ABB RobotStudio station: Robot Manipulatin Assignment 2 task 2.rspag

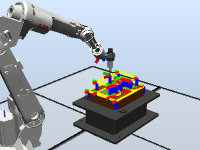
--- station ---
Station try1 (saved by RobotStudio 6.8.8148.134)
Controller IRB_1520ID_4kg_1.50m
  mechanical unit ROB_1: IRB1520ID_4_150__02, 6 joints, base frame (0, 0, 0) mm
Layout (positions relative to the parent item):
  - IRB1520ID_4_150__02 [mechanism, from Robots\IRB1520ID_4_150_G_02.rslib] at (0, 0, 0) mm; joint values [-0.2556, -0.3637, 0.7959, 0.3224, 0.5136, -0.4862] (rad or m)
  - MyTool [mechanism, from Training Objects\myTool.rslib] at (791.12, -174.55, 725.53) mm, rotated rx 180 ry 38 rz 180 deg
  - Robotpedestal1400_H240 [part, from Equipment\Robot Pedestal 1400 H240.rslib] at (1106.08, -98.58, 0) mm
  - Curve_thing [part, from Training Objects\Curve_Thing.rslib] at (902, -245, 225) mm
  - Frame_1 [frame] at (902, -245, 225) mm
Attachment: MyTool is attached to IRB1520ID_4_150__02 / Link6

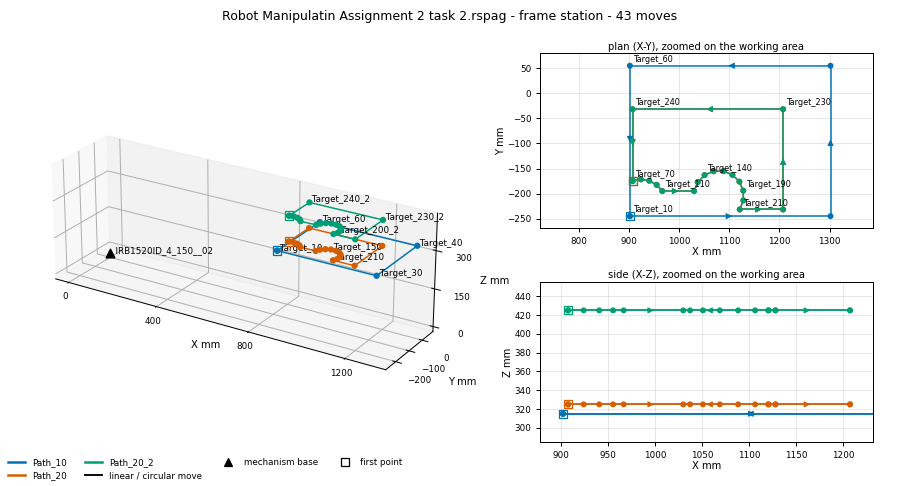
[picture p0: tool path of Robot Manipulatin Assignment 2 task 2.rspag in frame station, 43 of 49 moves have a stored position in this frame; points joined in program order, loops and branches not executed]
--- Backups/IRB_1520ID_4kg_1.50m/RAPID/TASK1/PROGMOD/CalibData.mod ---
MODULE CalibData
	PERS tooldata MyTool:=[TRUE,[[31.792631019,0,229.638935148],[0.945518576,0,0.325568154,0]],[1,[0,0,1],[1,0,0,0],0,0,0]];
ENDMODULE

--- Backups/IRB_1520ID_4kg_1.50m/RAPID/TASK1/PROGMOD/Module1.mod ---
MODULE Module1
    CONST robtarget Target_10:=[[901.999,-245.004,315],[0,0,1,0],[0,0,0,0],[9E+09,9E+09,9E+09,9E+09,9E+09,9E+09]];
    CONST robtarget Target_30:=[[1301.999,-245.004,315],[0,0,1,0],[0,0,0,0],[9E+09,9E+09,9E+09,9E+09,9E+09,9E+09]];
    CONST robtarget Target_40:=[[1301.999,54.996,315],[0,0,1,0],[0,0,0,0],[9E+09,9E+09,9E+09,9E+09,9E+09,9E+09]];
    CONST robtarget Target_60:=[[901.999,54.996,315],[0,0,1,0],[0,0,0,0],[9E+09,9E+09,9E+09,9E+09,9E+09,9E+09]];
    CONST robtarget Target_70:=[[907.446746826,-174.551583792,325],[0,0,1,0],[0,0,0,0],[9E+09,9E+09,9E+09,9E+09,9E+09,9E+09]];
    CONST robtarget Target_80:=[[924.004893302,-171.650689779,325],[0,0,1,0],[0,0,0,0],[9E+09,9E+09,9E+09,9E+09,9E+09,9E+09]];
    CONST robtarget Target_90:=[[940.588636002,-174.40148582,325],[0,0,1,0],[0,0,0,0],[9E+09,9E+09,9E+09,9E+09,9E+09,9E+09]];
    CONST robtarget Target_100:=[[955.323432229,-182.493035793,325],[0,0,1,0],[0,0,0,0],[9E+09,9E+09,9E+09,9E+09,9E+09,9E+09]];
    CONST robtarget Target_110:=[[966.543734874,-195.01071167,325],[0,0,1,0],[0,0,0,0],[9E+09,9E+09,9E+09,9E+09,9E+09,9E+09]];
    CONST robtarget Target_120:=[[1029.963932921,-195.01071167,325],[0,0,1,0],[0,0,0,0],[9E+09,9E+09,9E+09,9E+09,9E+09,9E+09]];
    CONST robtarget Target_130:=[[1037.281757518,-176.953168948,325],[0,0,1,0],[0,0,0,0],[9E+09,9E+09,9E+09,9E+09,9E+09,9E+09]];
    CONST robtarget Target_140:=[[1050.94577414,-163.063602514,325],[0,0,1,0],[0,0,0,0],[9E+09,9E+09,9E+09,9E+09,9E+09,9E+09]];
    CONST robtarget Target_150:=[[1068.881099643,-155.451145285,325],[0,0,1,0],[0,0,0,0],[9E+09,9E+09,9E+09,9E+09,9E+09,9E+09]];
    CONST robtarget Target_160:=[[1088.364251938,-155.271750128,325],[0,0,1,0],[0,0,0,0],[9E+09,9E+09,9E+09,9E+09,9E+09,9E+09]];
    CONST robtarget Target_170:=[[1106.436711185,-162.552658227,325],[0,0,1,0],[0,0,0,0],[9E+09,9E+09,9E+09,9E+09,9E+09,9E+09]];
    CONST robtarget Target_180:=[[1120.354171512,-176.188262505,325],[0,0,1,0],[0,0,0,0],[9E+09,9E+09,9E+09,9E+09,9E+09,9E+09]];
    CONST robtarget Target_190:=[[1128.003264309,-194.107994237,325],[0,0,1,0],[0,0,0,0],[9E+09,9E+09,9E+09,9E+09,9E+09,9E+09]];
    CONST robtarget Target_200:=[[1128.222473592,-213.59073925,325],[0,0,1,0],[0,0,0,0],[9E+09,9E+09,9E+09,9E+09,9E+09,9E+09]];
    CONST robtarget Target_210:=[[1120.978512397,-231.678039551,325],[0,0,1,0],[0,0,0,0],[9E+09,9E+09,9E+09,9E+09,9E+09,9E+09]];
    CONST robtarget Target_220:=[[1207.446746826,-231.678039551,325],[0,0,1,0],[0,0,0,0],[9E+09,9E+09,9E+09,9E+09,9E+09,9E+09]];
    CONST robtarget Target_230:=[[1207.446746826,-31.678039551,325],[0,0,1,0],[0,0,0,0],[9E+09,9E+09,9E+09,9E+09,9E+09,9E+09]];
    CONST robtarget Target_240:=[[907.446746826,-31.678039551,325],[0,0,1,0],[0,0,0,0],[9E+09,9E+09,9E+09,9E+09,9E+09,9E+09]];
    CONST robtarget Target_10_2:=[[901.999,-245.004,415],[0,0,1,0],[0,0,0,0],[9E+09,9E+09,9E+09,9E+09,9E+09,9E+09]];
    CONST robtarget Target_30_2:=[[1301.999,-245.004,415],[0,0,1,0],[0,0,0,0],[9E+09,9E+09,9E+09,9E+09,9E+09,9E+09]];
    CONST robtarget Target_40_2:=[[1301.999,54.996,415],[0,0,1,0],[0,0,0,0],[9E+09,9E+09,9E+09,9E+09,9E+09,9E+09]];
    CONST robtarget Target_60_2:=[[901.999,54.996,415],[0,0,1,0],[0,0,0,0],[9E+09,9E+09,9E+09,9E+09,9E+09,9E+09]];
    CONST robtarget Target_70_2:=[[907.446746826,-174.551583792,425],[0,0,1,0],[0,0,0,0],[9E+09,9E+09,9E+09,9E+09,9E+09,9E+09]];
    CONST robtarget Target_80_2:=[[924.004893302,-171.650689779,425],[0,0,1,0],[0,0,0,0],[9E+09,9E+09,9E+09,9E+09,9E+09,9E+09]];
    CONST robtarget Target_90_2:=[[940.588636002,-174.40148582,425],[0,0,1,0],[0,0,0,0],[9E+09,9E+09,9E+09,9E+09,9E+09,9E+09]];
    CONST robtarget Target_100_2:=[[955.323432229,-182.493035793,425],[0,0,1,0],[0,0,0,0],[9E+09,9E+09,9E+09,9E+09,9E+09,9E+09]];
    CONST robtarget Target_110_2:=[[966.543734874,-195.01071167,425],[0,0,1,0],[0,0,0,0],[9E+09,9E+09,9E+09,9E+09,9E+09,9E+09]];
    CONST robtarget Target_120_2:=[[1029.963932921,-195.01071167,425],[0,0,1,0],[0,0,0,0],[9E+09,9E+09,9E+09,9E+09,9E+09,9E+09]];
    CONST robtarget Target_130_2:=[[1037.281757518,-176.953168948,425],[0,0,1,0],[0,0,0,0],[9E+09,9E+09,9E+09,9E+09,9E+09,9E+09]];
    CONST robtarget Target_140_2:=[[1050.94577414,-163.063602514,425],[0,0,1,0],[0,0,0,0],[9E+09,9E+09,9E+09,9E+09,9E+09,9E+09]];
    CONST robtarget Target_150_2:=[[1068.881099643,-155.451145285,425],[0,0,1,0],[0,0,0,0],[9E+09,9E+09,9E+09,9E+09,9E+09,9E+09]];
    CONST robtarget Target_160_2:=[[1088.364251938,-155.271750128,425],[0,0,1,0],[0,0,0,0],[9E+09,9E+09,9E+09,9E+09,9E+09,9E+09]];
    CONST robtarget Target_170_2:=[[1106.436711185,-162.552658227,425],[0,0,1,0],[0,0,0,0],[9E+09,9E+09,9E+09,9E+09,9E+09,9E+09]];
    CONST robtarget Target_180_2:=[[1120.354171512,-176.188262505,425],[0,0,1,0],[0,0,0,0],[9E+09,9E+09,9E+09,9E+09,9E+09,9E+09]];
    CONST robtarget Target_190_2:=[[1128.003264309,-194.107994237,425],[0,0,1,0],[0,0,0,0],[9E+09,9E+09,9E+09,9E+09,9E+09,9E+09]];
    CONST robtarget Target_200_2:=[[1128.222473592,-213.59073925,425],[0,0,1,0],[0,0,0,0],[9E+09,9E+09,9E+09,9E+09,9E+09,9E+09]];
    CONST robtarget Target_210_2:=[[1120.978512397,-231.678039551,425],[0,0,1,0],[0,0,0,0],[9E+09,9E+09,9E+09,9E+09,9E+09,9E+09]];
    CONST robtarget Target_220_2:=[[1207.446746826,-231.678039551,425],[0,0,1,0],[0,0,0,0],[9E+09,9E+09,9E+09,9E+09,9E+09,9E+09]];
    CONST robtarget Target_230_2:=[[1207.446746826,-31.678039551,425],[0,0,1,0],[0,0,0,0],[9E+09,9E+09,9E+09,9E+09,9E+09,9E+09]];
    CONST robtarget Target_240_2:=[[907.446746826,-31.678039551,425],[0,0,1,0],[0,0,0,0],[9E+09,9E+09,9E+09,9E+09,9E+09,9E+09]];

    !Group #4 Assignment #2 Task #1

    PROC main()
        Path_10; !Initial workpiece platform welding
        Path_20; !Initial workpiece welding
        WaitTime 3; !3 seconds is the ETA of the new workpiece
        Path_20_2; !Posterior workpiece welding
    ENDPROC

    PROC Path_10() !Initial workpiece platform welding
        VAR  robtarget Target_10_prime;
        Target_10_prime:=Offs(Target_10,0,0,50); !This is an offset point with respect Prior_Target (Prior_Target,X,Y,Z)
        !up to the actual point then we straight go down to that point by the robot. This is the assignment requirement
        MoveJ Target_10_prime,v300,z100,MyTool\WObj:=wobj0; !The first point with joint movement to provide the robot flexibility
        MoveL Target_10,v300,z100,MyTool\WObj:=wobj0; !The rest using linear movement set the velocity to v=300 and zone point z=fine as for welding tasks precission is required
        MoveL Target_30,v300,fine,MyTool\WObj:=wobj0;
        MoveL Target_40,v300,fine,MyTool\WObj:=wobj0;
        MoveL Target_60,v300,fine,MyTool\WObj:=wobj0;
        MoveL Target_10,v300,fine,MyTool\WObj:=wobj0;
        MoveL Target_10_prime,v300,z100,MyTool\WObj:=wobj0;
    ENDPROC
    PROC Path_20() !Initial workpiece welding
        VAR  robtarget Target_70_prime;
        Target_70_prime:=Offs(Target_70,0,0,150);
        MoveJ Target_70_prime,v300,z100,MyTool\WObj:=wobj0;
        MoveL Target_70,v300,fine,MyTool\WObj:=wobj0;
        MoveL Target_80,v300,fine,MyTool\WObj:=wobj0;
        MoveL Target_90,v300,fine,MyTool\WObj:=wobj0;
        MoveL Target_100,v300,fine,MyTool\WObj:=wobj0;
        MoveL Target_110,v300,fine,MyTool\WObj:=wobj0;
        MoveL Target_120,v300,fine,MyTool\WObj:=wobj0;
        MoveL Target_130,v300,fine,MyTool\WObj:=wobj0;
        MoveL Target_140,v300,fine,MyTool\WObj:=wobj0;
        MoveL Target_150,v300,fine,MyTool\WObj:=wobj0;
        MoveL Target_160,v300,fine,MyTool\WObj:=wobj0;
        MoveL Target_170,v300,fine,MyTool\WObj:=wobj0;
        MoveL Target_180,v300,fine,MyTool\WObj:=wobj0;
        MoveL Target_190,v300,fine,MyTool\WObj:=wobj0;
        MoveL Target_200,v300,fine,MyTool\WObj:=wobj0;
        MoveL Target_210,v300,fine,MyTool\WObj:=wobj0;
        MoveL Target_220,v300,fine,MyTool\WObj:=wobj0;
        MoveL Target_230,v300,fine,MyTool\WObj:=wobj0;
        MoveL Target_240,v300,fine,MyTool\WObj:=wobj0;
        MoveL Target_70,v300,fine,MyTool\WObj:=wobj0;
        MoveL Target_70_prime,v300,z100,MyTool\WObj:=wobj0;
    ENDPROC
    PROC Path_20_2() !Posterior workpiece welding
        VAR  robtarget Target_70_prime2;
        Target_70_prime2:=Offs(Target_70_2,0,0,100);
        MoveJ Target_70_prime2,v300,z100,MyTool\WObj:=wobj0;
        MoveL Target_70_2,v300,fine,MyTool\WObj:=wobj0;
        MoveL Target_80_2,v300,fine,MyTool\WObj:=wobj0;
        MoveL Target_90_2,v300,fine,MyTool\WObj:=wobj0;
        MoveL Target_100_2,v300,fine,MyTool\WObj:=wobj0;
        MoveL Target_110_2,v300,fine,MyTool\WObj:=wobj0;
        MoveL Target_120_2,v300,fine,MyTool\WObj:=wobj0;
        MoveL Target_130_2,v300,fine,MyTool\WObj:=wobj0;
        MoveL Target_140_2,v300,fine,MyTool\WObj:=wobj0;
        MoveL Target_150_2,v300,fine,MyTool\WObj:=wobj0;
        MoveL Target_160_2,v300,fine,MyTool\WObj:=wobj0;
        MoveL Target_170_2,v300,fine,MyTool\WObj:=wobj0;
        MoveL Target_180_2,v300,fine,MyTool\WObj:=wobj0;
        MoveL Target_190_2,v300,fine,MyTool\WObj:=wobj0;
        MoveL Target_200_2,v300,fine,MyTool\WObj:=wobj0;
        MoveL Target_210_2,v300,fine,MyTool\WObj:=wobj0;
        MoveL Target_220_2,v300,fine,MyTool\WObj:=wobj0;
        MoveL Target_230_2,v300,fine,MyTool\WObj:=wobj0;
        MoveL Target_240_2,v300,fine,MyTool\WObj:=wobj0;
        MoveL Target_70_2,v300,fine,MyTool\WObj:=wobj0;
        MoveL Target_70_prime2,v300,z100,MyTool\WObj:=wobj0;
    ENDPROC
ENDMODULE

--- Backups/IRB_1520ID_4kg_1.50m/RAPID/TASK1/PROGMOD/RsTempModule.mod ---
MODULE RsTempModule
PROC RsTempPath()
ENDPROC

ENDMODULE

--- Backups/IRB_1520ID_4kg_1.50m/RAPID/TASK1/SYSMOD/LINKEDM.sys ---
%%%
  VERSION:1
  LANGUAGE:ENGLISH
%%%

MODULE LINKEDM (SYSMODULE)

! FOLLOWER
!     Name of electronically linked follower axis used by operator at teach pendent.
      PERS string l_f_axis_name{5}       :=  ["",  "", "", "", ""];

!     Name of the mechanical unit for follower axis.
      PERS string l_f_mecunt_n{5}  :=  ["", "", "", "", ""];

!     Linked follower axis number in the mechanical unit (first axis in mech. unit is number 1).
      PERS num l_f_axis_no{5}      :=  [0,          0,   0,  0,  0];

! MASTER
!     Name of the mechanical unit for linked master axis.
      PERS string l_m_mecunt_n{5} :=  ["", "", "", "", ""];

!     Linked master axis number in the mechanical unit (first axis in mech. unit is number 1).
!     See axis number table in documentation for different master mechanical units.
      PERS num l_m_axis_no{5}     :=  [0,  0,  0,  0,  0];

! POSITION OFFSET
!     The increase of the allowed offset position between the master and follower
!     positions, used when starting AUTO mode. As soon as the offset is decreased
!     the old configurated parameter is used.
!     Example: 3 => the configurated value of allowed offset is increased 3 times.
      PERS num offset_ratio{5}       :=  [10,  10,   10,  10,  10];

! SPEED RATIO
!     Speed_ratio used in AUTO and JOG modes [ very_slow   slow    normal    fast]
!     Value 1 = max allowed manual speed.
      CONST num speed_ratio {20}      := [0.01, 0.01, 0.01, 0.01, 0.01,
                                          0.05, 0.05, 0.05, 0.05, 0.05,
                                          0.20, 0.20, 0.20, 0.20, 0.20,
                                          1.00, 1.00, 1.00, 1.00, 1.00];

! STEP SIZE
!     Displacement position used in JOG mode for each activation of positive or
!     negative movement.                  [very_short    short   normal   long]
!     Unit degees or meter.
      CONST num displacement {20}     := [0.001, 0.001, 0.001, 0.001, 0.001,
                                          0.005, 0.005, 0.005, 0.005, 0.005,
                                          0.020, 0.020, 0.020, 0.020, 0.020,
                                          0.100, 0.100, 0.100, 0.100, 0.100];


!-------------------------------------------------------------
 PROC Linked_m ()
      Linked_m_exe ;
 ENDPROC
ENDMODULE
